{attribute addProperty BoxType "EK1122-0000-0018"}
{attribute addProperty Id "Beckhoff_EL7xxxsub_EK1100EK1100_179A0949162"}
{attribute addProperty CRC "3562659407"}
{attribute addProperty SizeInBites "16"}
{attribute addProperty SizeInBytes "2"}
TYPE Beckhoff_EL7xxxEK1122_D459DE4F EXTENDS EK1122_179A0949 :
STRUCT
	{attribute addProperty Name "Beckhoff_EL7xxxsub_EK1100"}
	Beckhoff_EL7xxxsub_EK1100 : EK1100_179A0949;
END_STRUCT
END_TYPE

(* stored: Version 1.2.0.0, ProductVersion 3.1.4024.9
   DUT Beckhoff_EL7xxxEK1122_D459DE4F: Id {3680199c-5f93-4af2-877c-767788b59315} *)
